// SIMATIC S7-200 project (STEP 7-Micro/WIN), CPU 226 REL 02.01

SYMBOL_TABLE MESSAGES
STATUS_MESSAGE   VB1000   // Target for status messages
FIVE_VOLT_MESSAGE VB1080
YELLOW_BUTTON1_MESSAGE VB1120
YELLOW_BUTTON2_MESSAGE VB1160
ESTOP_MESSAGE    VB1200
FAULT_MESSAGE    VB1240
POWER_MESSAGE    VB1280
READY_MESSAGE    VB1320
PC_READY_MESSAGE VB1360
END_SYMBOL_TABLE

SYMBOL_TABLE USS Protocol
USS_LOW_V        VD1000   // (DWORD) Enter the starting address for USS Protocol symbols here.
USS_HIGH_V       VD1004
USS_TIME_OUT     VW1008
USS_I_LINE       VW1010
USS_DAT_PTR0     VD1012
USS_ACT_DRV0     VD1016
USS_CUR_DRV0     VD1020
USS_P0           V1024.0
USS_REQ_SNT0     V1024.1
USS_RETRY_P0     VB1025
USS_ERR_CODE     VB1026
USS_CS_D0        VD1027
USS_CS_W0        VW1027
USS_CS_W2        VW1029
USS_CS_B0        VB1027
USS_CS_B1        VB1028
USS_POLL_BUF     VB1031
USS_XMT_0        VB1046
USS_XMT_ADR0     VB1049
USS_X_STWD       VD1056
USS_X_BCC        VB1060
USS_X_DW1        VD1047
USS_X_DW5        VD1051
USS_X_DW9        VD1055
USS_X_DB13       VB1059
USS_RCV_BUF0     VB1061
USS_R_STX        VB1062
USS_R_LGE        VB1063
USS_R_ADR        VB1064
USS_R_STWD       VD1071
USS_R_DW1        VD1062
USS_R_DW5        VD1066
USS_R_DW9        VD1070
USS_R_W13        VW1074
USS_STAT_TAB     VB1076
USS_ADR_P0       VB1396
END_SYMBOL_TABLE

SYMBOL_TABLE PC
INNER_HALT_PC    I0.0     // INNER Motor HALT
INNER_VELOCITY_MODE_PC I0.1     // CUST INNER STEP/VEL SWITCH
OUTER_VELOCITY_MODE_PC I0.2     // CUST OUTER POS/VEL SWITCH
OUTER_HALT_PC    I0.3     // PIitch Motor HALT
PC_READY         I0.6     // PC Ready
HMI_ALARM        Q1.3     // Notify PC of alarm(s)
PLC_OK           Q1.2     // PLC OK to PC
END_SYMBOL_TABLE

SYMBOL_TABLE OUTER
OUTER_VELOCITY_RAW AIW8     // OUTER VELOCITY FEEDBACK
OUTER_TORQUE_RAW AIW10    // OUTER TORQUE FEEDBACK
OUTER_COMMAND_RAW AIW12    // OUTER VELOCITY RATE COMMAND
OUTER_Z_PUSLE    I1.1     // OUTER I/REV
OUTER_MSP_OVERLOAD I1.7     // OUTER OVERLOAD
OUTER_RELAY_FEEDBACK I2.0     // OUTER BB
OUTER_DRIVE_READY I2.5     // OUTER Controller READY
OUTER_MOTOR_RDY  I2.6     // OUTER Motor READY
OUTER_DRIVE_WARNING I2.7     // OUTER WARNING
OUTER_LOCK       I3.0     // OUTER MANUALLY LOCKED
OUTER_SERVO_READY M4.3     // OUTER Drive Ready to Operate
OUTER_MODE       MB10     // OUTER Mode
OUTER_POWER      Q0.0     // OUTER Control Power
OUTER_POSITION_MODE Q1.6     // OUTER STEP POS OUT
OUTER_ENABLE     Q2.0     // OUTER ENABLE
OUTER_ESTOP      Q2.1     // OUTER E-STOP
OUTER_CLEAR_ERROR Q2.2     // OUTER CLEAR ERROR
OUTER_DYNAMIC_BRAKE Q2.3     // OUTER DYNAMIC BRAKE
OUTER_HALT       Q2.4     // OUTER HALT
OUTER_HOME       Q2.5     // OUTER HOME START
OUTER_VELOCITY_MODE Q2.6     // OUTER STEP/VEL MODE SWOTCH
OUTER_POWER_DELAY T38      // OUTER CONTROL DELAY
OUTER_DYN_BRAKE_DELAY T39      // OUTER DYNAMIC  BRAKE DELAY
OUTER_TORQUE_HIGH_DELAY T41      // OUTER TORQUE HIGH
OUTER_ERROR_DELAY T42      // OUTER DC BUS FAULT DELAY
OUTER_SERVO_DELAY T45      // OUTER SERVO DELAY
OUTER_BRAKE_DELAY T46      // OUTER BRAKE DELAY
OUTER_VELOCITY   VD1428
OUTER_TORQUE     VD1472
OUTER_COMMAND    VD1476
OUTER_VELOCITY_M VD1480
OUTER_VELOCITY_B VD1484
OUTER_TORQUE_M   VD1488
OUTER_TORQUE_B   VD1492
OUTER_COMMAND_M  VD1496
OUTER_COMMAND_B  VD1500
END_SYMBOL_TABLE

SYMBOL_TABLE INNER
INNER_VELOCITY_RAW AIW0     // INNER VELOCITY FEEDBACK
INNER_TORQUE_RAW AIW2     // INNER TORQUE FEEDBACK
INNER_COMMAND_RAW AIW4     // INNER VELOCITY RATE COMMAND
INNER_Z_PULSE    I1.0     // INNER 1/REV
INNER_MSP_OVERLOAD I1.5     // MSP OVERLOAD INNER MOTOR
INNER_RELAY_FEEDBACK I1.6     // INNER Master Control Relay (CR910) Auxiliary Contact
INNER_DRIVE_READY I2.2     // INNER Controller READY
INNER_MOTOR_READY I2.3     // INNER MOTOR READY
INNER_DRIVE_WARNING I2.4     // INNER Drive WARNING
INNER_COMMUTATE  M4.4     // INNER Drive Commutation Mode
INNER_SERVO_READY M0.3     // INNER Drive Ready to Operate
INNER_MODE       MB9      // INNER Mode
INNER_POWER      Q0.1     // INNER Control Power
INNER_ENABLE     Q0.2     // INNER Drive ENABLE
INNER_ESTOP      Q0.3     // INNER Emergency Stop
INNER_CLEAR_ERROR Q0.4     // INNER Drive Clear Error
INNER_DYNAMIC_BRAKE Q0.5     // INNER DYNAMIC BRAKE
INNER_HALT       Q0.6     // INNER Motor HOLD ON/OFF
INNER_HOME       Q0.7     // INNER START HOME
INNER_VELOCITY_MODE Q1.0     // INNER VELOCITY MODE  SELECT
INNER_POSITION_MODE Q1.7     // INNER POSITION
INNER_POWER_DELAY T33      // K1 DELAY
INNER_DYN_BRAKE_DELAY T34      // INNER Dynamic Brake Delay
INNER_ERROR_DELAY T37      // INNER DC BUS FAULT DELAY
INNER_TORQUE_HIGH_DELAY T40      // INNER TORQUE TOO HIGH
INNER_SERVO_DELAY T47      // INNER Servo Controller Delay
INNER_BRAKE_DELAY T48      // INNER Brake Delay
INNER_VELOCITY   VD428
INNER_TORQUE     VD472
INNER_COMMAND    VD476
INNER_VELOCITY_M VD480
INNER_VELOCITY_B VD484
INNER_TORQUE_M   VD488
INNER_TORQUE_B   VD492
INNER_COMMAND_M  VD496
INNER_COMMAND_B  VD500
END_SYMBOL_TABLE

SYMBOL_TABLE INTERLOC
WARNING_LEFT     I1.2     // PATIENT WARNING LEFT
WARNING_RIGHT    I1.3     // PATIENT WARNING RIGHT
MAIN_POWER_SIGNAL I1.4     // Main Power Signal
ESTOP            I2.1     // Emergency Stop
TWO_AXIS_BRAKE_1 I3.1     // TWO AXIS BRAKE FROM PB
SEAT_BELT_INTERLOCK I3.2     // SEAT BELT INTERLOCK
FIVE_VOLT_INTERLOCK I3.3     // EXTRA FIVE VOLT CLOSURE INTERLOCK
TWO_AXIS_BRAKE_2 I3.4     // Second 2-axis brake from pushbutton
AREA_SAFE        M7.6     // Area safe bit
GREEN_ALLCLEAR_LIGHT Q1.5     // Green Allclear Light
RED_WARNING_LIGHT Q2.7     // Red Warning Light
MINIMUM_ESTOP_DELAY T36      // Minimum ESTOP fault duration delay
AREA_SAFE_TIMER  T49      // Area Safe Timer
MASTER_FAULT     M0.2     // Master Fault
PB_BRAKE         M7.1     // PB TWO AXIS BRAKE
HALT_LEVEL_FAULT M11.1    // Faults that don't de-energize the motors
END_SYMBOL_TABLE

SYMBOL_TABLE LABELS
NO_MORE_MESSAGES_LABEL 1        // End of messages section
SKIP_POWER_DEP_FAULTS 2
END_SYMBOL_TABLE

SYMBOL_TABLE HMI
RESET            M0.5     // Reset
DYNAMIC_BRAKE_SUSPEND M1.0     // Dynamic Brake Suspend (from HMI)
INNER_HALT_HMI   M2.3     // INNER HALT BUTTON (HMI)
OUTER_HALT_HMI   M4.5     // OUTER Brake Release PB (HMI)
HMI_MODE         MB8      // HMIMode
SWITCH_ON_NOT_RED_FAULT V6.0     // SWITCH ON WITHOUT RED LIGHT FAULT
OUTER_OVERLOAD_FAULT V6.1     // OUTER MSP1 OVERLOAD
OUTER_ERROR_FAULT V6.2     // OUTER ERROR FAULT BIT
MAIN_POWER_FAULT V6.5     // Main Power Fault Bit
OUTER_COMMAND_FAULT V6.6     // OUTER COMMAND TOO HIGH
OUTER_VELOCITY_FAULT V6.7     // OUTER VELOCITY TOO HIGH
INNER_OVERLOAD_FAULT V7.0     // INNER MOTOR STARTER PROTECTOR (MSP2) OVERLOAD
ESTOP_FAULT      V7.1     // Emergency Stop Bit
INNER_ERROR_FAULT V7.2     // INNER ERROR FAULT
OUTER_LOCK_FAULT V7.4     // Outer axis lock fault bit
INNER_COMMAND_FAULT V7.5     // INNER RATE COMMAND TOO HIGH
INNER_VELOCITY_FAULT V7.6     // INNER VELOCITY HIGH
INNER_TORQUE_FAULT V7.7     // INNER TORQUE HIIGH
FIVE_VOLT_FAULT  V8.0     // 5V safety closure fault bit
OUTER_WARNING_FAULT V8.1     // OUTER MOTOR WARNING
OUTER_TORQUE_FAULT V9.1     // OUTER TORQUE TOO HIGH BIT
INNER_WARNING_FAULT V9.2     // INNER MOTOR WARNING
DATE_AND_TIME    VB10     // PLC Date and Time for HMI
END_SYMBOL_TABLE

SYMBOL_TABLE RESERVED
RESERVED         Q1.1     // Reserved (Do Not Use)
END_SYMBOL_TABLE

SYMBOL_TABLE TEMPORARY
D_TMP            MD16
END_SYMBOL_TABLE

ORGANIZATION_BLOCK Program_Block:OB1
TITLE=Brandeis University
// HULK/PRY/TARC - AFOSR
// Author: Neuro Kinetics Inc., Ashton Graybiel Spatial Orientation Laboratory
// Date: May 2007
BEGIN
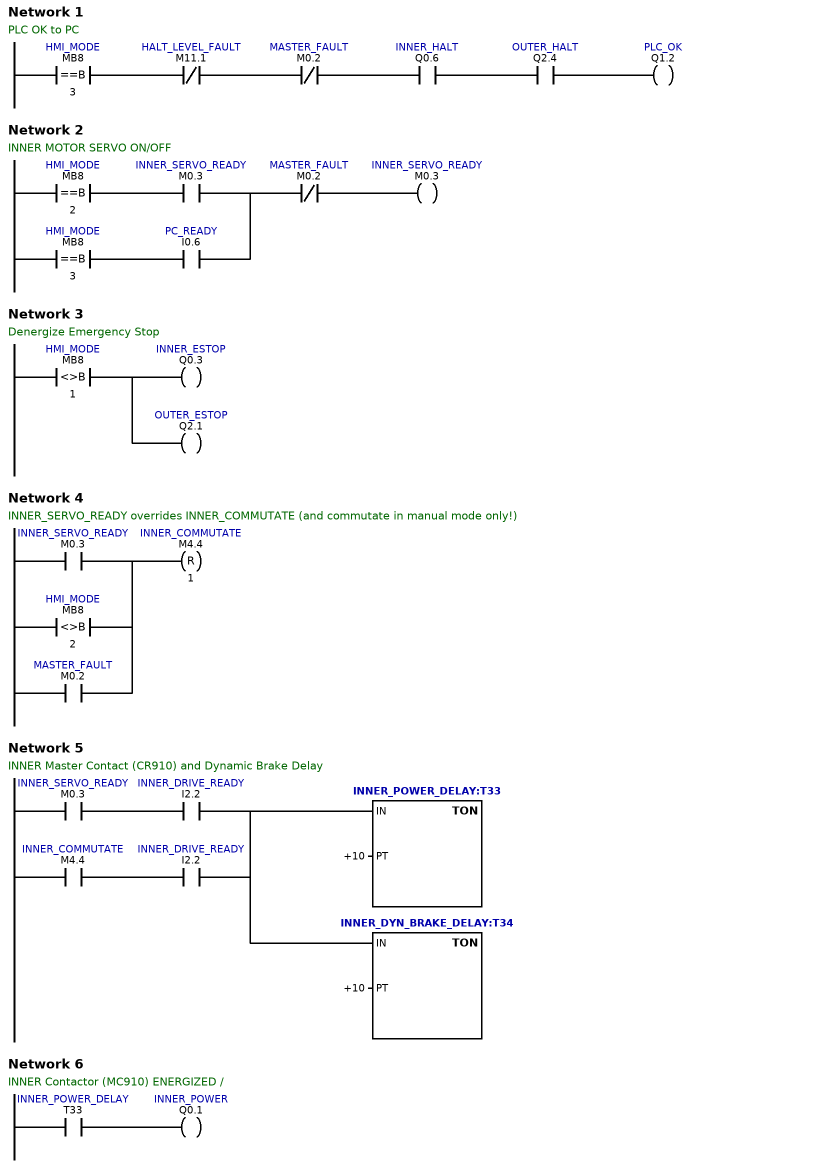
Network 1
// PLC OK to PC
LDB=   HMI_MODE:MB8, 3
AN     HALT_LEVEL_FAULT:M11.1
AN     MASTER_FAULT:M0.2
A      INNER_HALT:Q0.6
A      OUTER_HALT:Q2.4
=      PLC_OK:Q1.2
Network 2
//  INNER MOTOR SERVO ON/OFF
LDB=   HMI_MODE:MB8, 2
A      INNER_SERVO_READY:M0.3
LDB=   HMI_MODE:MB8, 3
A      PC_READY:I0.6
OLD
AN     MASTER_FAULT:M0.2
=      INNER_SERVO_READY:M0.3
Network 3
// Denergize Emergency Stop
LDB<>  HMI_MODE:MB8, 1
=      INNER_ESTOP:Q0.3
=      OUTER_ESTOP:Q2.1
Network 4
// INNER_SERVO_READY overrides INNER_COMMUTATE (and commutate in manual mode only!)
LD     INNER_SERVO_READY:M0.3
OB<>   HMI_MODE:MB8, 2
O      MASTER_FAULT:M0.2
R      INNER_COMMUTATE:M4.4, 1
Network 5
// INNER Master Contact (CR910) and Dynamic Brake Delay
LD     INNER_SERVO_READY:M0.3
A      INNER_DRIVE_READY:I2.2
LD     INNER_COMMUTATE:M4.4
A      INNER_DRIVE_READY:I2.2
OLD
TON    INNER_POWER_DELAY:T33, +10
TON    INNER_DYN_BRAKE_DELAY:T34, +10
Network 6
// INNER Contactor (MC910) ENERGIZED
// 
LD     INNER_POWER_DELAY:T33
=      INNER_POWER:Q0.1
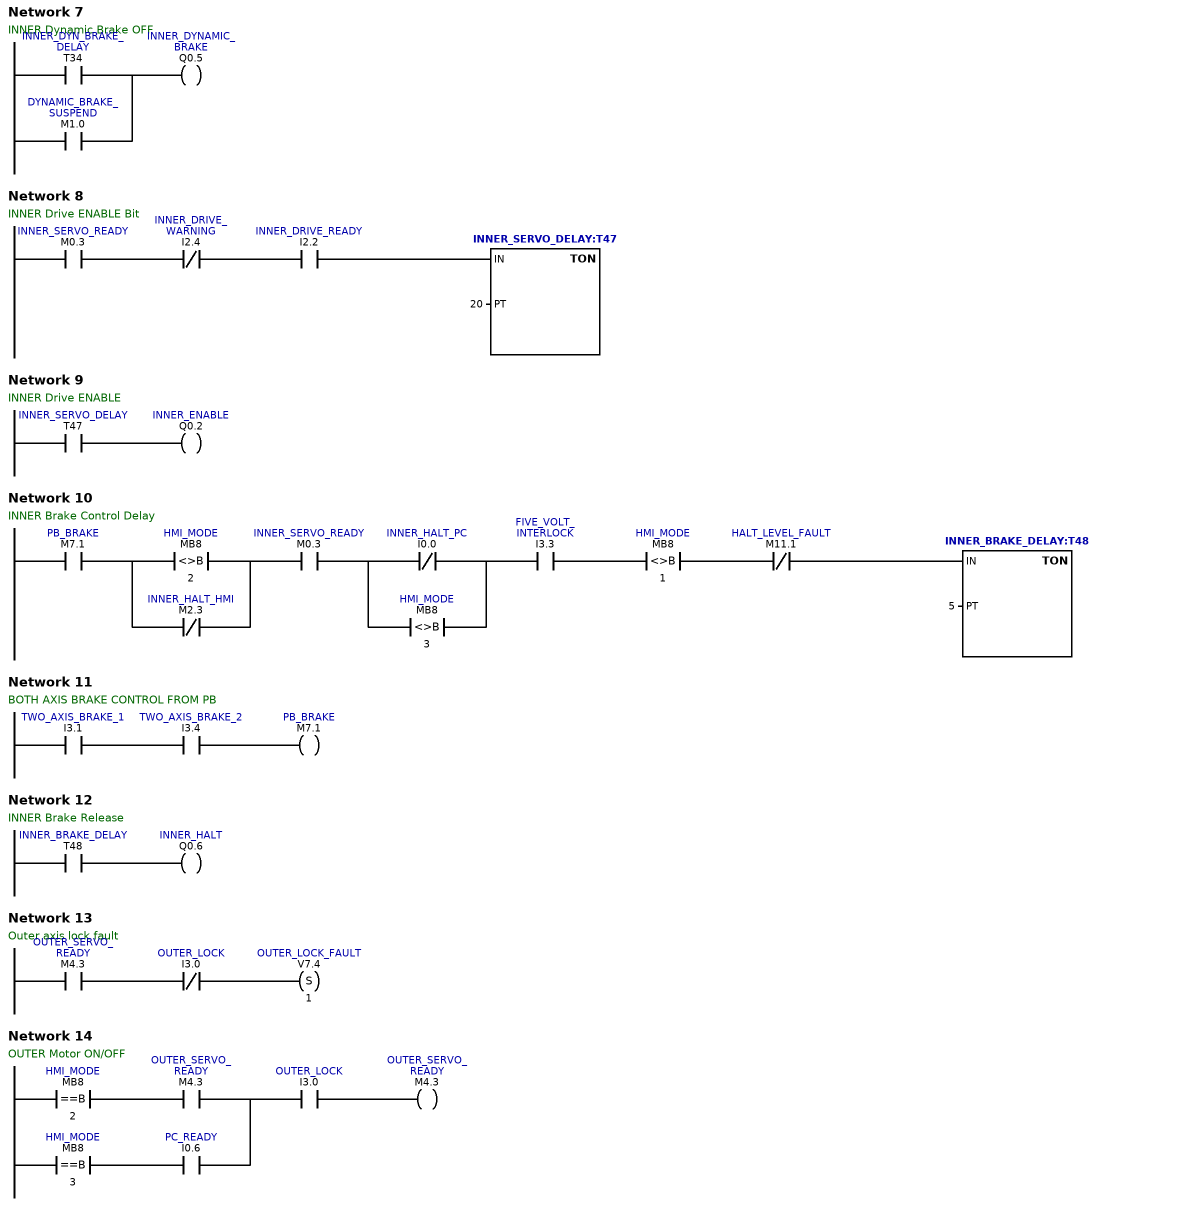
Network 7
// INNER Dynamic Brake OFF
LD     INNER_DYN_BRAKE_DELAY:T34
O      DYNAMIC_BRAKE_SUSPEND:M1.0
=      INNER_DYNAMIC_BRAKE:Q0.5
Network 8
// INNER Drive ENABLE Bit
LD     INNER_SERVO_READY:M0.3
AN     INNER_DRIVE_WARNING:I2.4
A      INNER_DRIVE_READY:I2.2
TON    INNER_SERVO_DELAY:T47, 20
Network 9
// INNER Drive ENABLE
LD     INNER_SERVO_DELAY:T47
=      INNER_ENABLE:Q0.2
Network 10
// INNER Brake Control Delay
LD     PB_BRAKE:M7.1
LDB<>  HMI_MODE:MB8, 2
ON     INNER_HALT_HMI:M2.3
ALD
A      INNER_SERVO_READY:M0.3
LDN    INNER_HALT_PC:I0.0
OB<>   HMI_MODE:MB8, 3
ALD
A      FIVE_VOLT_INTERLOCK:I3.3
AB<>   HMI_MODE:MB8, 1
AN     HALT_LEVEL_FAULT:M11.1
TON    INNER_BRAKE_DELAY:T48, 5
Network 11
// BOTH AXIS BRAKE CONTROL FROM PB
LD     TWO_AXIS_BRAKE_1:I3.1
A      TWO_AXIS_BRAKE_2:I3.4
=      PB_BRAKE:M7.1
Network 12
// INNER Brake Release
LD     INNER_BRAKE_DELAY:T48
=      INNER_HALT:Q0.6
Network 13
// Outer axis lock fault
LD     OUTER_SERVO_READY:M4.3
AN     OUTER_LOCK:I3.0
S      OUTER_LOCK_FAULT:V7.4, 1
Network 14
//  OUTER Motor ON/OFF
LDB=   HMI_MODE:MB8, 2
A      OUTER_SERVO_READY:M4.3
LDB=   HMI_MODE:MB8, 3
A      PC_READY:I0.6
OLD
A      OUTER_LOCK:I3.0
=      OUTER_SERVO_READY:M4.3
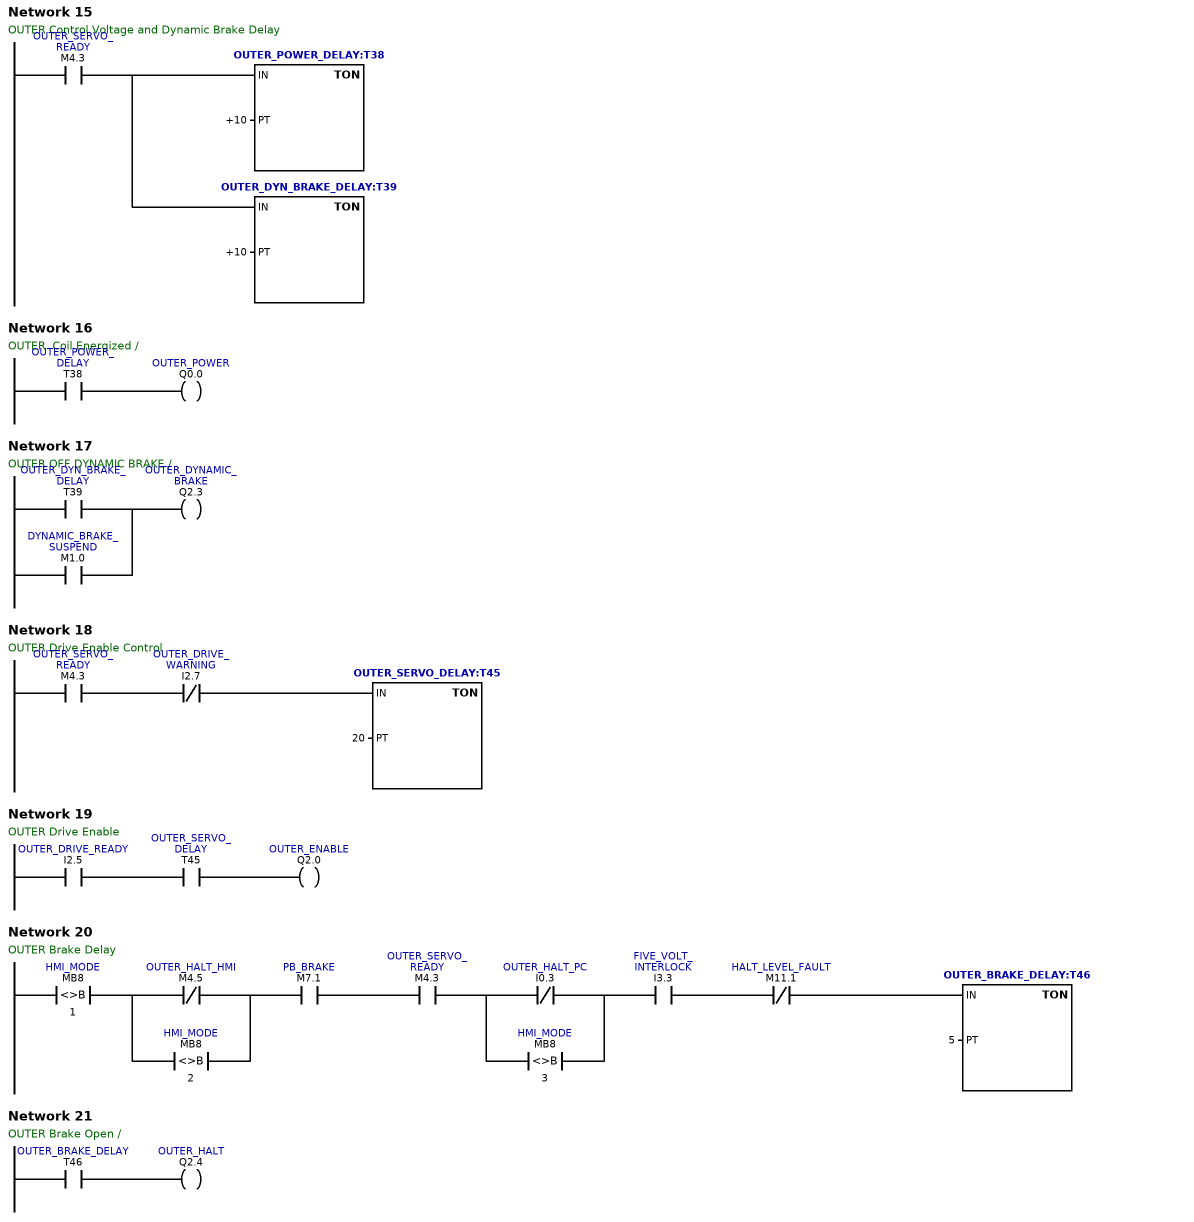
Network 15
// OUTER Control Voltage and Dynamic Brake Delay
LD     OUTER_SERVO_READY:M4.3
TON    OUTER_POWER_DELAY:T38, +10
TON    OUTER_DYN_BRAKE_DELAY:T39, +10
Network 16
// OUTER  Coil Energized
// 
LD     OUTER_POWER_DELAY:T38
=      OUTER_POWER:Q0.0
Network 17
// OUTER OFF DYNAMIC BRAKE
// 
LD     OUTER_DYN_BRAKE_DELAY:T39
O      DYNAMIC_BRAKE_SUSPEND:M1.0
=      OUTER_DYNAMIC_BRAKE:Q2.3
Network 18
// OUTER Drive Enable Control
LD     OUTER_SERVO_READY:M4.3
AN     OUTER_DRIVE_WARNING:I2.7
TON    OUTER_SERVO_DELAY:T45, 20
Network 19
// OUTER Drive Enable
LD     OUTER_DRIVE_READY:I2.5
A      OUTER_SERVO_DELAY:T45
=      OUTER_ENABLE:Q2.0
Network 20
// OUTER Brake Delay
LDB<>  HMI_MODE:MB8, 1
LDN    OUTER_HALT_HMI:M4.5
OB<>   HMI_MODE:MB8, 2
ALD
A      PB_BRAKE:M7.1
A      OUTER_SERVO_READY:M4.3
LDN    OUTER_HALT_PC:I0.3
OB<>   HMI_MODE:MB8, 3
ALD
A      FIVE_VOLT_INTERLOCK:I3.3
AN     HALT_LEVEL_FAULT:M11.1
TON    OUTER_BRAKE_DELAY:T46, 5
Network 21
// OUTER Brake Open
// 
LD     OUTER_BRAKE_DELAY:T46
=      OUTER_HALT:Q2.4
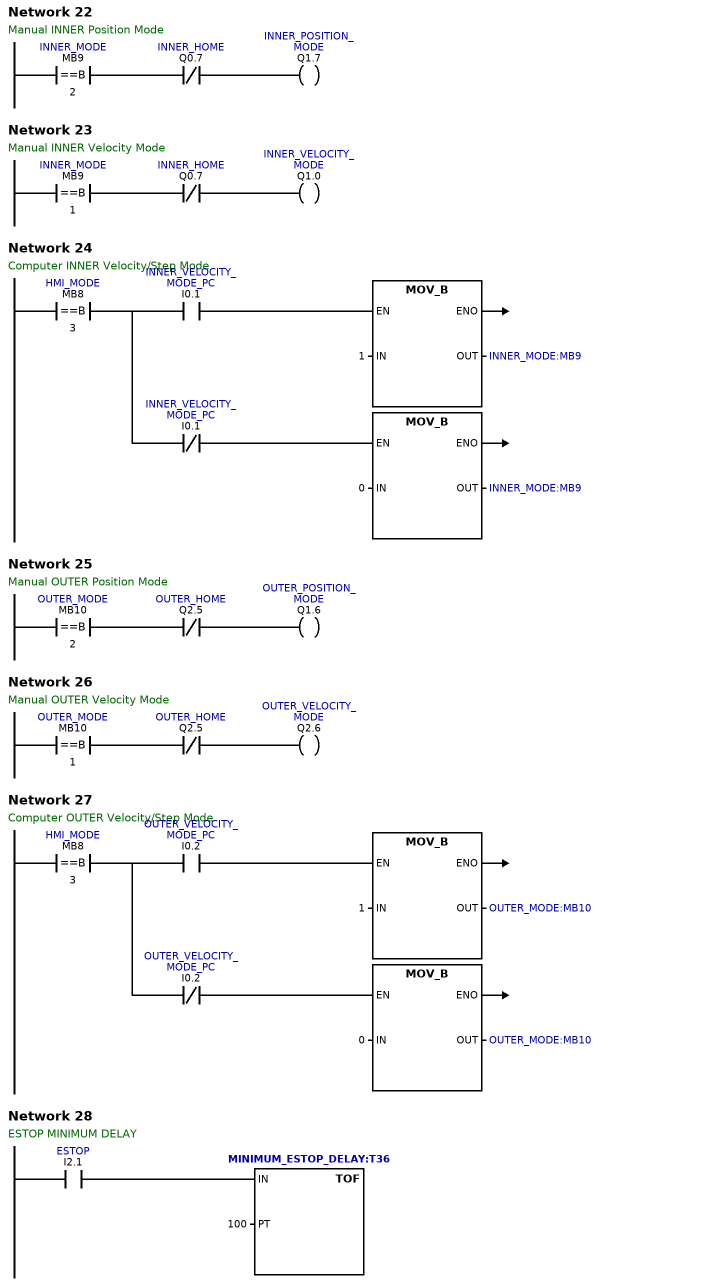
Network 22
// Manual INNER Position Mode
LDB=   INNER_MODE:MB9, 2
AN     INNER_HOME:Q0.7
=      INNER_POSITION_MODE:Q1.7
Network 23
// Manual INNER Velocity Mode
LDB=   INNER_MODE:MB9, 1
AN     INNER_HOME:Q0.7
=      INNER_VELOCITY_MODE:Q1.0
Network 24
// Computer INNER Velocity/Step Mode
LDB=   HMI_MODE:MB8, 3
LPS
A      INNER_VELOCITY_MODE_PC:I0.1
MOVB   1, INNER_MODE:MB9
LPP
AN     INNER_VELOCITY_MODE_PC:I0.1
MOVB   0, INNER_MODE:MB9
Network 25
// Manual OUTER Position Mode
LDB=   OUTER_MODE:MB10, 2
AN     OUTER_HOME:Q2.5
=      OUTER_POSITION_MODE:Q1.6
Network 26
// Manual OUTER Velocity Mode
LDB=   OUTER_MODE:MB10, 1
AN     OUTER_HOME:Q2.5
=      OUTER_VELOCITY_MODE:Q2.6
Network 27
// Computer OUTER Velocity/Step Mode
LDB=   HMI_MODE:MB8, 3
LPS
A      OUTER_VELOCITY_MODE_PC:I0.2
MOVB   1, OUTER_MODE:MB10
LPP
AN     OUTER_VELOCITY_MODE_PC:I0.2
MOVB   0, OUTER_MODE:MB10
Network 28
// ESTOP MINIMUM DELAY
LD     ESTOP:I2.1
TOF    MINIMUM_ESTOP_DELAY:T36, 100
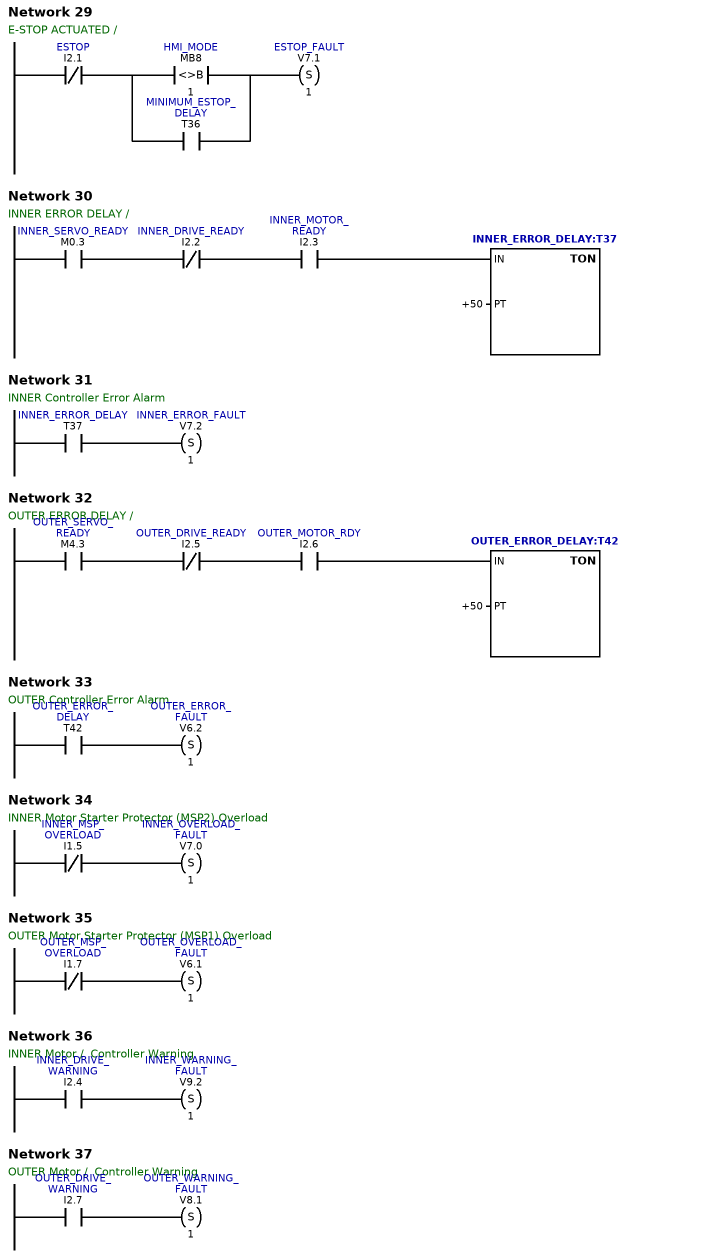
Network 29
// E-STOP ACTUATED
// 
LDN    ESTOP:I2.1
LDB<>  HMI_MODE:MB8, 1
O      MINIMUM_ESTOP_DELAY:T36
ALD
S      ESTOP_FAULT:V7.1, 1
Network 30
// INNER ERROR DELAY
// 
LD     INNER_SERVO_READY:M0.3
AN     INNER_DRIVE_READY:I2.2
A      INNER_MOTOR_READY:I2.3
TON    INNER_ERROR_DELAY:T37, +50
Network 31
// INNER Controller Error Alarm
LD     INNER_ERROR_DELAY:T37
S      INNER_ERROR_FAULT:V7.2, 1
Network 32
// OUTER ERROR DELAY
// 
LD     OUTER_SERVO_READY:M4.3
AN     OUTER_DRIVE_READY:I2.5
A      OUTER_MOTOR_RDY:I2.6
TON    OUTER_ERROR_DELAY:T42, +50
Network 33
// OUTER Controller Error Alarm
LD     OUTER_ERROR_DELAY:T42
S      OUTER_ERROR_FAULT:V6.2, 1
Network 34
// INNER Motor Starter Protector (MSP2) Overload
LDN    INNER_MSP_OVERLOAD:I1.5
S      INNER_OVERLOAD_FAULT:V7.0, 1
Network 35
// OUTER Motor Starter Protector (MSP1) Overload
LDN    OUTER_MSP_OVERLOAD:I1.7
S      OUTER_OVERLOAD_FAULT:V6.1, 1
Network 36
// INNER Motor /  Controller Warning
LD     INNER_DRIVE_WARNING:I2.4
S      INNER_WARNING_FAULT:V9.2, 1
Network 37
// OUTER Motor /  Controller Warning
LD     OUTER_DRIVE_WARNING:I2.7
S      OUTER_WARNING_FAULT:V8.1, 1
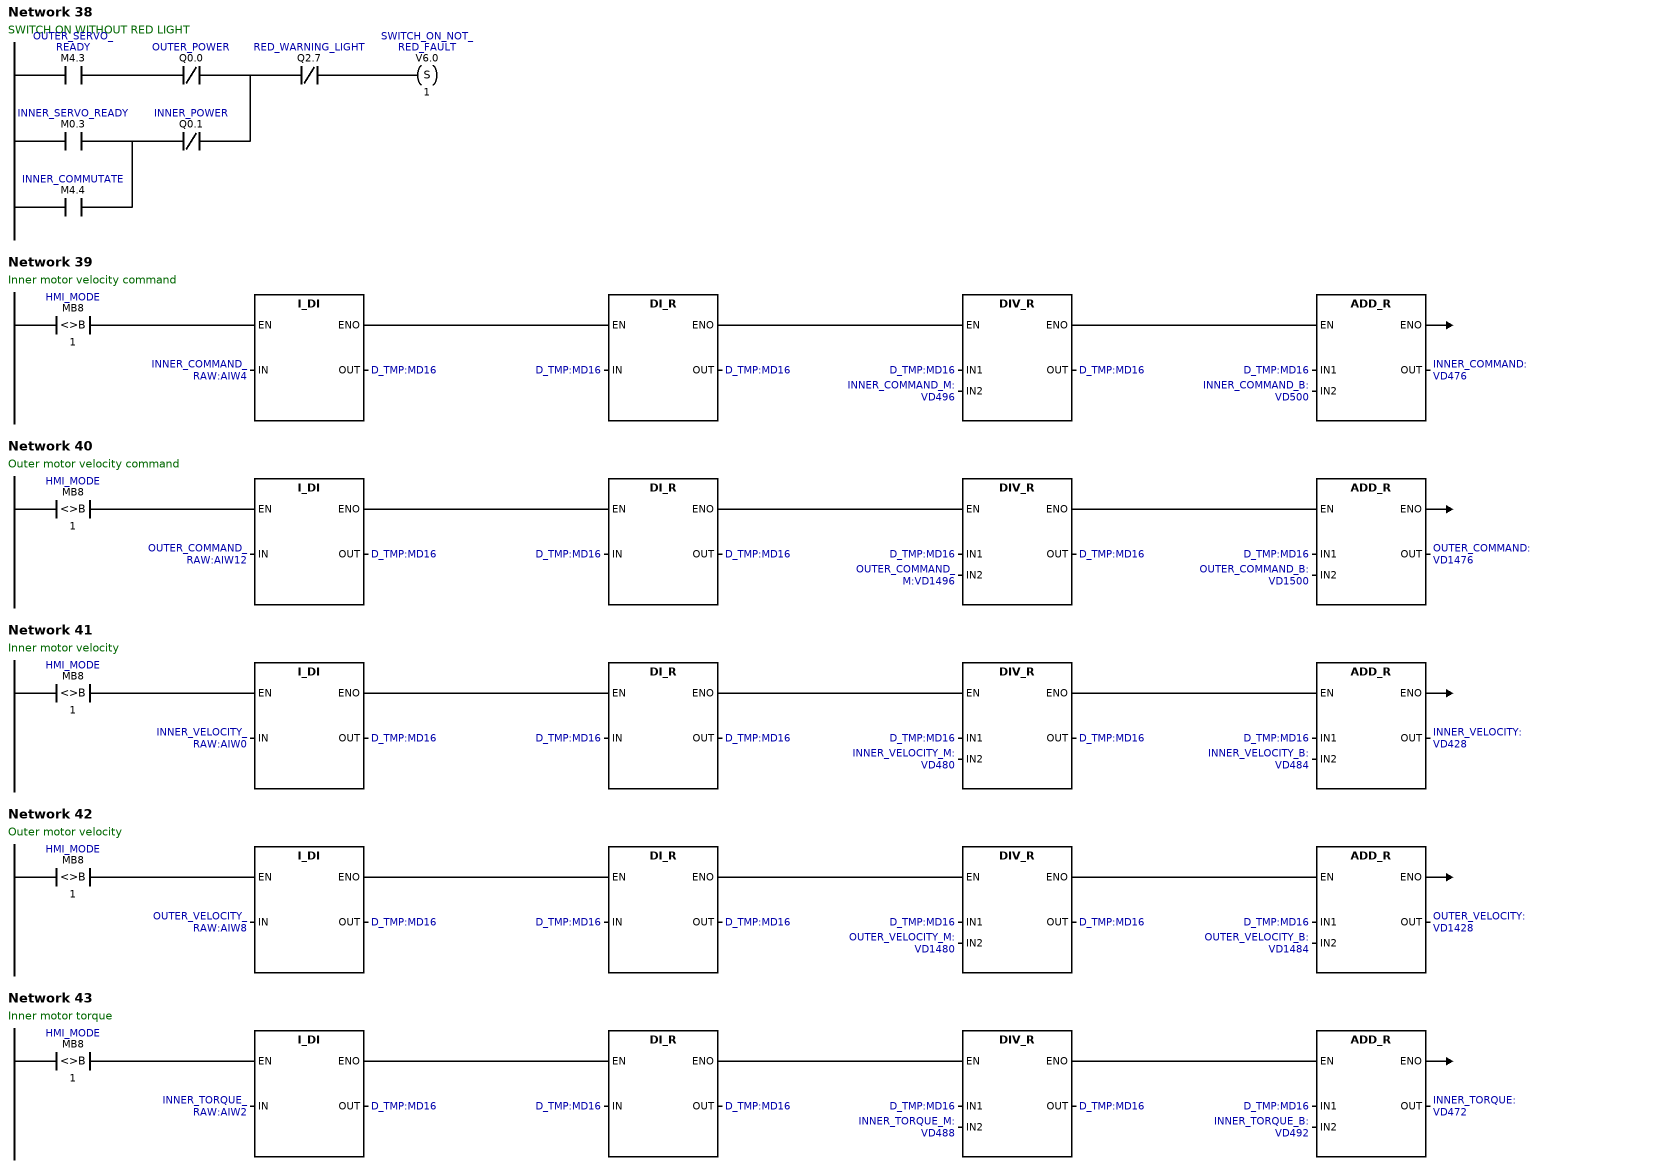
Network 38
// SWITCH ON WITHOUT RED LIGHT
LD     OUTER_SERVO_READY:M4.3
AN     OUTER_POWER:Q0.0
LD     INNER_SERVO_READY:M0.3
O      INNER_COMMUTATE:M4.4
AN     INNER_POWER:Q0.1
OLD
AN     RED_WARNING_LIGHT:Q2.7
S      SWITCH_ON_NOT_RED_FAULT:V6.0, 1
Network 39
// Inner motor velocity command
LDB<>  HMI_MODE:MB8, 1
ITD    INNER_COMMAND_RAW:AIW4, D_TMP:MD16
AENO
DTR    D_TMP:MD16, D_TMP:MD16
AENO
/R     INNER_COMMAND_M:VD496, D_TMP:MD16
AENO
MOVR   D_TMP:MD16, INNER_COMMAND:VD476
+R     INNER_COMMAND_B:VD500, INNER_COMMAND:VD476
Network 40
// Outer motor velocity command
LDB<>  HMI_MODE:MB8, 1
ITD    OUTER_COMMAND_RAW:AIW12, D_TMP:MD16
AENO
DTR    D_TMP:MD16, D_TMP:MD16
AENO
/R     OUTER_COMMAND_M:VD1496, D_TMP:MD16
AENO
MOVR   D_TMP:MD16, OUTER_COMMAND:VD1476
+R     OUTER_COMMAND_B:VD1500, OUTER_COMMAND:VD1476
Network 41
// Inner motor velocity
LDB<>  HMI_MODE:MB8, 1
ITD    INNER_VELOCITY_RAW:AIW0, D_TMP:MD16
AENO
DTR    D_TMP:MD16, D_TMP:MD16
AENO
/R     INNER_VELOCITY_M:VD480, D_TMP:MD16
AENO
MOVR   D_TMP:MD16, INNER_VELOCITY:VD428
+R     INNER_VELOCITY_B:VD484, INNER_VELOCITY:VD428
Network 42
// Outer motor velocity
LDB<>  HMI_MODE:MB8, 1
ITD    OUTER_VELOCITY_RAW:AIW8, D_TMP:MD16
AENO
DTR    D_TMP:MD16, D_TMP:MD16
AENO
/R     OUTER_VELOCITY_M:VD1480, D_TMP:MD16
AENO
MOVR   D_TMP:MD16, OUTER_VELOCITY:VD1428
+R     OUTER_VELOCITY_B:VD1484, OUTER_VELOCITY:VD1428
Network 43
// Inner motor torque
LDB<>  HMI_MODE:MB8, 1
ITD    INNER_TORQUE_RAW:AIW2, D_TMP:MD16
AENO
DTR    D_TMP:MD16, D_TMP:MD16
AENO
/R     INNER_TORQUE_M:VD488, D_TMP:MD16
AENO
MOVR   D_TMP:MD16, INNER_TORQUE:VD472
+R     INNER_TORQUE_B:VD492, INNER_TORQUE:VD472
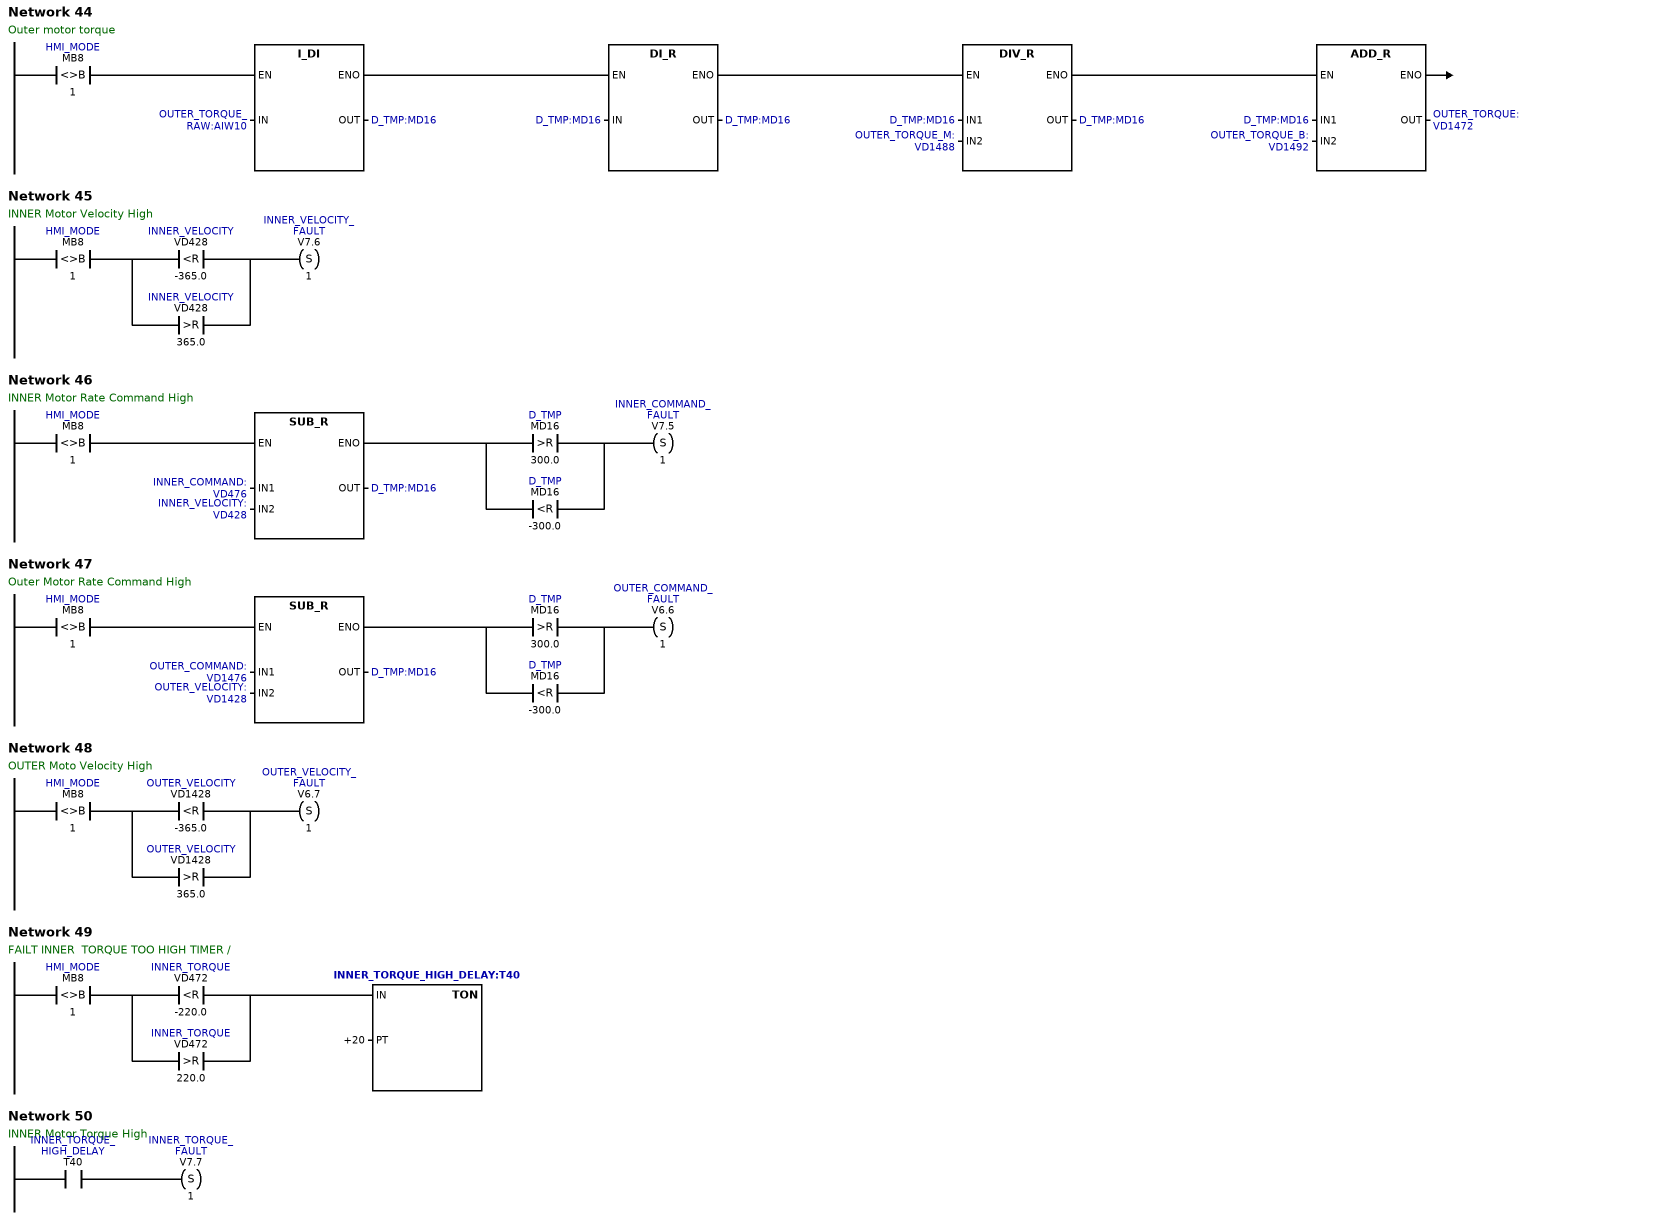
Network 44
// Outer motor torque
LDB<>  HMI_MODE:MB8, 1
ITD    OUTER_TORQUE_RAW:AIW10, D_TMP:MD16
AENO
DTR    D_TMP:MD16, D_TMP:MD16
AENO
/R     OUTER_TORQUE_M:VD1488, D_TMP:MD16
AENO
MOVR   D_TMP:MD16, OUTER_TORQUE:VD1472
+R     OUTER_TORQUE_B:VD1492, OUTER_TORQUE:VD1472
Network 45
// INNER Motor Velocity High
LDB<>  HMI_MODE:MB8, 1
LDR<   INNER_VELOCITY:VD428, -365.0
OR>    INNER_VELOCITY:VD428, 365.0
ALD
S      INNER_VELOCITY_FAULT:V7.6, 1
Network 46
// INNER Motor Rate Command High
LDB<>  HMI_MODE:MB8, 1
MOVR   INNER_COMMAND:VD476, D_TMP:MD16
AENO
-R     INNER_VELOCITY:VD428, D_TMP:MD16
AENO
LDR>   D_TMP:MD16, 300.0
OR<    D_TMP:MD16, -300.0
ALD
S      INNER_COMMAND_FAULT:V7.5, 1
Network 47
// Outer Motor Rate Command High
LDB<>  HMI_MODE:MB8, 1
MOVR   OUTER_COMMAND:VD1476, D_TMP:MD16
AENO
-R     OUTER_VELOCITY:VD1428, D_TMP:MD16
AENO
LDR>   D_TMP:MD16, 300.0
OR<    D_TMP:MD16, -300.0
ALD
S      OUTER_COMMAND_FAULT:V6.6, 1
Network 48
// OUTER Moto Velocity High
LDB<>  HMI_MODE:MB8, 1
LDR<   OUTER_VELOCITY:VD1428, -365.0
OR>    OUTER_VELOCITY:VD1428, 365.0
ALD
S      OUTER_VELOCITY_FAULT:V6.7, 1
Network 49
// FAILT INNER  TORQUE TOO HIGH TIMER
// 
LDB<>  HMI_MODE:MB8, 1
LDR<   INNER_TORQUE:VD472, -220.0
OR>    INNER_TORQUE:VD472, 220.0
ALD
TON    INNER_TORQUE_HIGH_DELAY:T40, +20
Network 50
// INNER Motor Torque High
LD     INNER_TORQUE_HIGH_DELAY:T40
S      INNER_TORQUE_FAULT:V7.7, 1
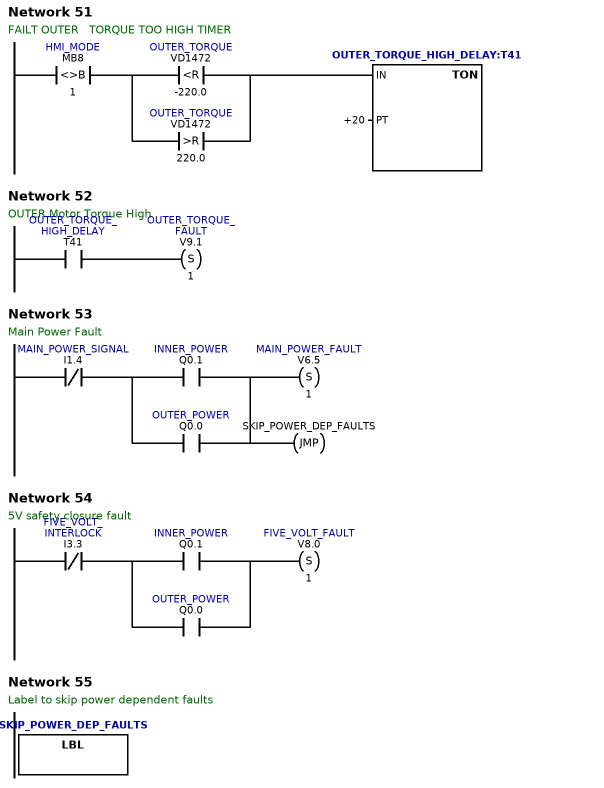
Network 51
// FAILT OUTER   TORQUE TOO HIGH TIMER
LDB<>  HMI_MODE:MB8, 1
LDR<   OUTER_TORQUE:VD1472, -220.0
OR>    OUTER_TORQUE:VD1472, 220.0
ALD
TON    OUTER_TORQUE_HIGH_DELAY:T41, +20
Network 52
// OUTER Motor Torque High
LD     OUTER_TORQUE_HIGH_DELAY:T41
S      OUTER_TORQUE_FAULT:V9.1, 1
Network 53
// Main Power Fault
LDN    MAIN_POWER_SIGNAL:I1.4
LD     INNER_POWER:Q0.1
O      OUTER_POWER:Q0.0
ALD
S      MAIN_POWER_FAULT:V6.5, 1
JMP    SKIP_POWER_DEP_FAULTS
Network 54
// 5V safety closure fault
LDN    FIVE_VOLT_INTERLOCK:I3.3
LD     INNER_POWER:Q0.1
O      OUTER_POWER:Q0.0
ALD
S      FIVE_VOLT_FAULT:V8.0, 1
Network 55
// Label to skip power dependent faults
LBL    SKIP_POWER_DEP_FAULTS
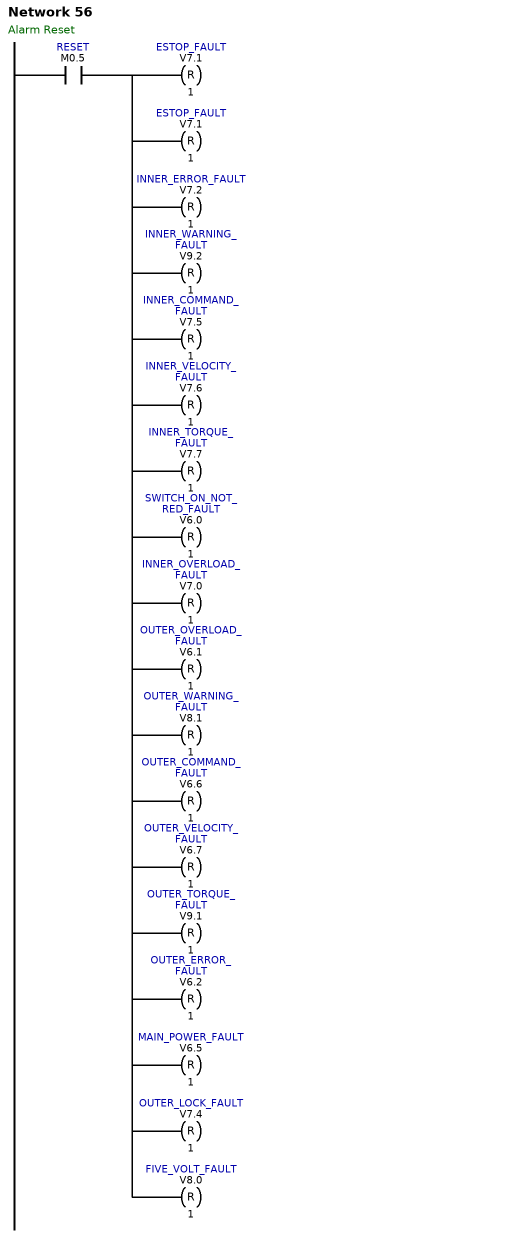
Network 56
// Alarm Reset
LD     RESET:M0.5
R      ESTOP_FAULT:V7.1, 1
R      ESTOP_FAULT:V7.1, 1
R      INNER_ERROR_FAULT:V7.2, 1
R      INNER_WARNING_FAULT:V9.2, 1
R      INNER_COMMAND_FAULT:V7.5, 1
R      INNER_VELOCITY_FAULT:V7.6, 1
R      INNER_TORQUE_FAULT:V7.7, 1
R      SWITCH_ON_NOT_RED_FAULT:V6.0, 1
R      INNER_OVERLOAD_FAULT:V7.0, 1
R      OUTER_OVERLOAD_FAULT:V6.1, 1
R      OUTER_WARNING_FAULT:V8.1, 1
R      OUTER_COMMAND_FAULT:V6.6, 1
R      OUTER_VELOCITY_FAULT:V6.7, 1
R      OUTER_TORQUE_FAULT:V9.1, 1
R      OUTER_ERROR_FAULT:V6.2, 1
R      MAIN_POWER_FAULT:V6.5, 1
R      OUTER_LOCK_FAULT:V7.4, 1
R      FIVE_VOLT_FAULT:V8.0, 1
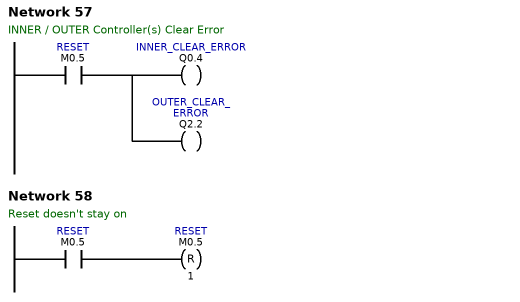
Network 57
// INNER / OUTER Controller(s) Clear Error
LD     RESET:M0.5
=      INNER_CLEAR_ERROR:Q0.4
=      OUTER_CLEAR_ERROR:Q2.2
Network 58
// Reset doesn't stay on
LD     RESET:M0.5
R      RESET:M0.5, 1
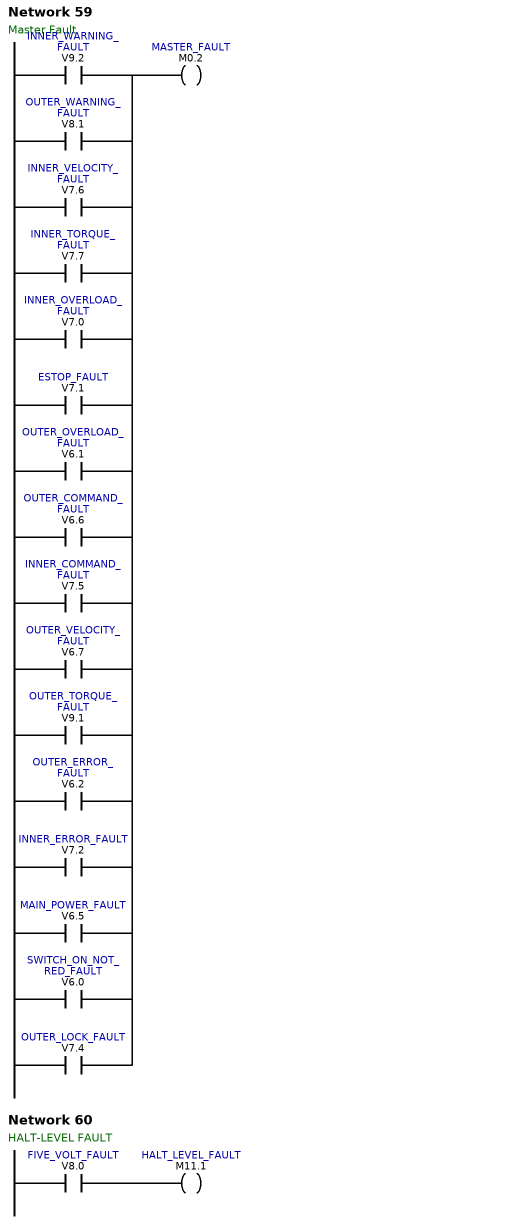
Network 59
// Master Fault
LD     INNER_WARNING_FAULT:V9.2
O      OUTER_WARNING_FAULT:V8.1
O      INNER_VELOCITY_FAULT:V7.6
O      INNER_TORQUE_FAULT:V7.7
O      INNER_OVERLOAD_FAULT:V7.0
O      ESTOP_FAULT:V7.1
O      OUTER_OVERLOAD_FAULT:V6.1
O      OUTER_COMMAND_FAULT:V6.6
O      INNER_COMMAND_FAULT:V7.5
O      OUTER_VELOCITY_FAULT:V6.7
O      OUTER_TORQUE_FAULT:V9.1
O      OUTER_ERROR_FAULT:V6.2
O      INNER_ERROR_FAULT:V7.2
O      MAIN_POWER_FAULT:V6.5
O      SWITCH_ON_NOT_RED_FAULT:V6.0
O      OUTER_LOCK_FAULT:V7.4
=      MASTER_FAULT:M0.2
Network 60
// HALT-LEVEL FAULT
LD     FIVE_VOLT_FAULT:V8.0
=      HALT_LEVEL_FAULT:M11.1
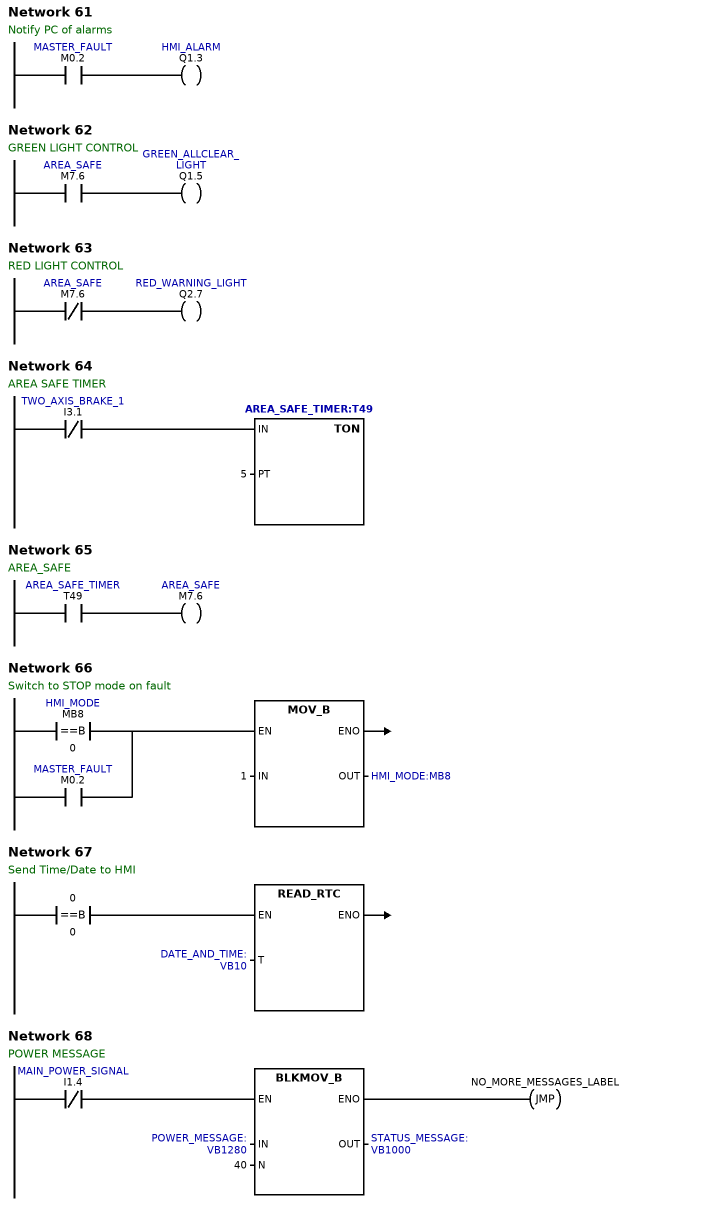
Network 61
// Notify PC of alarms
LD     MASTER_FAULT:M0.2
=      HMI_ALARM:Q1.3
Network 62
// GREEN LIGHT CONTROL
LD     AREA_SAFE:M7.6
=      GREEN_ALLCLEAR_LIGHT:Q1.5
Network 63
// RED LIGHT CONTROL
LDN    AREA_SAFE:M7.6
=      RED_WARNING_LIGHT:Q2.7
Network 64
// AREA SAFE TIMER
LDN    TWO_AXIS_BRAKE_1:I3.1
TON    AREA_SAFE_TIMER:T49, 5
Network 65
// AREA_SAFE
LD     AREA_SAFE_TIMER:T49
=      AREA_SAFE:M7.6
Network 66
// Switch to STOP mode on fault
LDB=   HMI_MODE:MB8, 0
O      MASTER_FAULT:M0.2
MOVB   1, HMI_MODE:MB8
Network 67
// Send Time/Date to HMI
LDB=   0, 0
TODR   DATE_AND_TIME:VB10
Network 68
// POWER MESSAGE
LDN    MAIN_POWER_SIGNAL:I1.4
BMB    POWER_MESSAGE:VB1280, STATUS_MESSAGE:VB1000, 40
AENO
JMP    NO_MORE_MESSAGES_LABEL
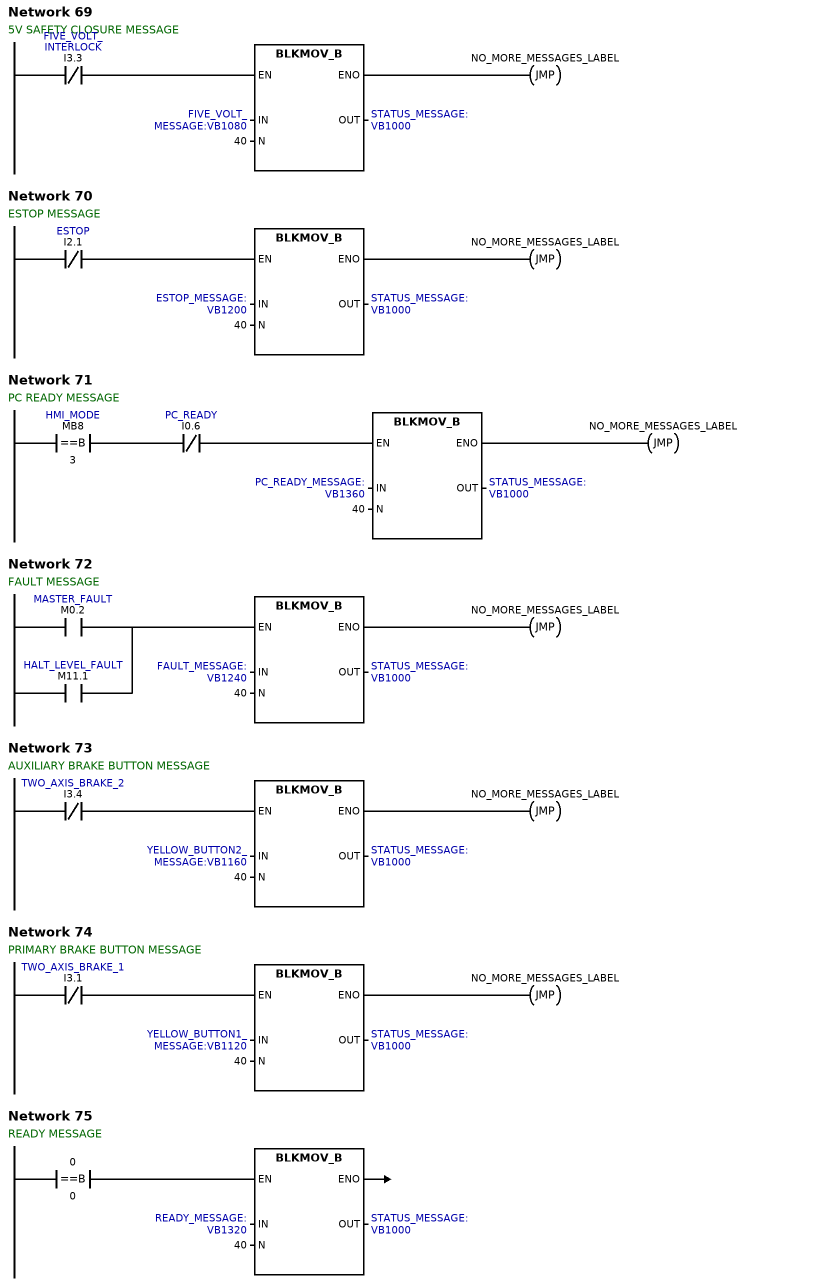
Network 69
// 5V SAFETY CLOSURE MESSAGE
LDN    FIVE_VOLT_INTERLOCK:I3.3
BMB    FIVE_VOLT_MESSAGE:VB1080, STATUS_MESSAGE:VB1000, 40
AENO
JMP    NO_MORE_MESSAGES_LABEL
Network 70
// ESTOP MESSAGE
LDN    ESTOP:I2.1
BMB    ESTOP_MESSAGE:VB1200, STATUS_MESSAGE:VB1000, 40
AENO
JMP    NO_MORE_MESSAGES_LABEL
Network 71
// PC READY MESSAGE
LDB=   HMI_MODE:MB8, 3
AN     PC_READY:I0.6
BMB    PC_READY_MESSAGE:VB1360, STATUS_MESSAGE:VB1000, 40
AENO
JMP    NO_MORE_MESSAGES_LABEL
Network 72
// FAULT MESSAGE
LD     MASTER_FAULT:M0.2
O      HALT_LEVEL_FAULT:M11.1
BMB    FAULT_MESSAGE:VB1240, STATUS_MESSAGE:VB1000, 40
AENO
JMP    NO_MORE_MESSAGES_LABEL
Network 73
// AUXILIARY BRAKE BUTTON MESSAGE
LDN    TWO_AXIS_BRAKE_2:I3.4
BMB    YELLOW_BUTTON2_MESSAGE:VB1160, STATUS_MESSAGE:VB1000, 40
AENO
JMP    NO_MORE_MESSAGES_LABEL
Network 74
// PRIMARY BRAKE BUTTON MESSAGE
LDN    TWO_AXIS_BRAKE_1:I3.1
BMB    YELLOW_BUTTON1_MESSAGE:VB1120, STATUS_MESSAGE:VB1000, 40
AENO
JMP    NO_MORE_MESSAGES_LABEL
Network 75
// READY MESSAGE
LDB=   0, 0
BMB    READY_MESSAGE:VB1320, STATUS_MESSAGE:VB1000, 40
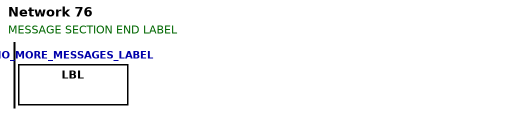
Network 76
// MESSAGE SECTION END LABEL
LBL    NO_MORE_MESSAGES_LABEL
END_ORGANIZATION_BLOCK

DATA_BLOCK_TAB MESSAGES
BEGIN
         READY_MESSAGE, 'READY'
         FAULT_MESSAGE, 'NOT READY: Unacknowledged fault'
         PC_READY_MESSAGE, 'NOT READY: No signal from PC'
         POWER_MESSAGE, 'NOT READY: Main power not detected'
         ESTOP_MESSAGE, 'NOT READY: Emergency stop button'
         YELLOW_BUTTON1_MESSAGE, 'NOT READY: Primary brake button'
         YELLOW_BUTTON2_MESSAGE, 'NOT READY: Auxiliary brake button'
         FIVE_VOLT_MESSAGE, 'NOT READY: 5V safety closure open'
END_DATA_BLOCK_TAB
